// TIA Portal V20 export
// export: Created 2025-12-01T14:57:04.2343757Z, ExportSetting None, DisplayName Totally Integrated Automation Portal, DisplayVersion V20 Update 3, DisplayName TIA Portal Openness, DisplayVersion V20 Update 3, DisplayName TIA Portal Version Control Interface, DisplayVersion V20 Update 3, DisplayName STEP 7 Professional, DisplayVersion V20 Update 3, DisplayName STEP 7 Safety, DisplayVersion V20 Update 2, DisplayName WinCC Basic/Comfort/Advanced, DisplayVersion V20 Update 3, DisplayName WinCC Professional, DisplayVersion V20 Update 3, DisplayName WinCC Unified, DisplayVersion V20 Update 3
FUNCTION "FC772_Control_ElevadorDobleHorq" : Void   // FC772, STL
TITLE = Tracking de la Maquina Base
{ S7_Optimized_Access := 'FALSE' }
AUTHOR : TRACKING
NAME : 20141014
VERSION : 4.0
// - Inicializar
// - Recoger datos necesarios del Sistema
// 
// - Dispositivo Maquina
//   + Gestion de Estado
//   + Gestion de Control de Reset
//   + Gestion de Control de Paro Blando
//   + Gestion de Control de Errores
// 
// - Operaciones propias de la Maquina
// 
// - Cierre de protocolo de la Maquina
// - Actualizar datos del Sistema
// stored: AutoNumber false
   VAR_INPUT
      EstadoZonaMaquina : "EstadoZona";   // Estado de la Maquina (ZONA)
      EstadoZonaMesaH01 : "EstadoZona";   // Estado de la Mesa H1 (ZONA)
      EstadoZonaMesaH02 : "EstadoZona";   // Estado de la Mesa H2 (ZONA)
      MaxPisos : UInt;   // Numero Maximo Pisos
      H01_Habilitada : Bool;   // Permiso trabajo con Horquilla 1
      H02_Habilitada : Bool;   // Permiso trabajo con Horquilla 2
      MesaH01_Vacia : Bool;   // Estado Mesa Horquilla 1 Vacia
      MesaH01_Cargada : Bool;   // Estado Mesa Horquilla 1 Cargada
      MesaH02_Vacia : Bool;   // Estado Mesa Horquilla 2 Vacia
      MesaH02_Cargada : Bool;   // Estado Mesa Horquilla 1 Cargada
      OrdenMesaH01 : Bool;   // Orden Tracking Mesa Horquilla 01
      OrdenMesaH02 : Bool;   // Orden Tracking Mesa Horquilla 02
      MesaDestinoH01 : UInt;   // Mesa Destino para UT en Mesa Horquilla 1
      MesaDestinoH02 : UInt;   // Mesa Destino para UT en Mesa Horquilla 2
      NDB_AuxliarElevador : UInt;   // Numero de DB auxiliar elevador
      OrdenH01_Acabada : Bool;   // Orden ejecutada por la Horquilla 1
      OrdenH02_Acabada : Bool;   // Orden ejecutada por la Horquilla 2
      OrdenPasarAReposo : Bool;   // Orden Para posicionar el carro en posición reposo
      PisoDeReposo : UInt;   // Piso para posición reposo
   END_VAR
   VAR_IN_OUT
      Orden_Piso : UInt;   // Piso del Movimiento a Ejecutar
      OrdenH01_TipoMovi : UInt;   // Tipo de Movimiento a Ejecutar con la Horquilla 1
      OrdenH02_TipoMovi : UInt;   // Tipo de Movimeinto a Ejecutar con la Horquilla 2
      MesaEntrada_H01 : UInt;   // Mesa con Transferencia hacia la Horquilla 1
      MesaEntrada_H02 : UInt;   // Mesa con Transferencia hacia la Horquilla 2
      MesaSalida_H01 : UInt;   // Mesa con Transferencia desde la Horquilla 1
      MesaSalida_H02 : UInt;   // Mesa con Transferencia desde la Horquilla 2
      OrdenH01_Realizar : Bool;   // Orden de Ejecutar Movimiento para la Horquilla 2
      OrdenH02_Realizar : Bool;   // Orden de Ejecutar Movimiento para la Horquilla 1
      MemoriaPisoCarga : UInt;   // Memoriza Ultimo Piso Carga
      PisoUltimaOrden : UInt;   // Memoriza Piso de la Ultima Orden Enviada
   END_VAR
   VAR_TEMP
      DBAuxElevador : Word;
      DBTMPTracking : Word;   // Num. DB de los Temporizadores
      Maquina : UInt;   // Numero de Maquina dentro del PLC
      NumPisoDescarga : UInt;
      TempInt : UInt;
      SinUT : Bool;
   END_VAR
BEGIN

NETWORK
TITLE = Inicializar
// - Inicializar las Varriables
// - Inicializar para la Base de datos
// - Inicializar para las comunicaciones
/////////////////////////////////////////////////////////////////////////////
// --- Inicializar las Variables



NETWORK
TITLE = Reset de Variables
/////////////////////////////////////////////////////////////////////////////
// --- Si realiza un reset hay que limpiar las variables

      AN    #EstadoZonaMaquina.PerReset_CBx;
      JC    NoExiste_Reset;  // Reseteada la Maquina

      L     0;  // Reseteo de las Ordenes de las Horquillas
      T     #OrdenH01_TipoMovi;
      T     #OrdenH02_TipoMovi;
      R     #OrdenH01_Realizar;
      R     #OrdenH02_Realizar;

      L     0;  // Reseteo del Numero de Piso
      T     #Orden_Piso;

      L     0;  // Datos del Tracking
      T     #MesaEntrada_H01;  // del elevador de doble Horquilla
      T     #MesaEntrada_H02;
      T     #MesaSalida_H01;
      T     #MesaSalida_H02;

      JU    FinalFuncion;  // Finalizado el tratamiento de la Maquina

NoExiste_Reset:NOP   0;



NETWORK
TITLE = Elevador Doble (Particular del Tipo de Maquina)
/////////////////////////////////////////////////////////////////////////////
// ---
// ---           GENERAR ORDNES PARA EL ELEVADOR DOBLE
// ---
/////////////////////////////////////////////////////////////////////////////

      L     #NDB_AuxliarElevador;  // DB Auxliar del Elevador
      T     #DBAuxElevador;


/////////////////////////////////////////////////////////////////////////////
// --- No Ordernes y alguna Vacia, incrementar piso, para buscar AVISO

      AN    #OrdenH01_Realizar;  // No tiene Orden H01
      AN    #OrdenH02_Realizar;  // No tiene Orden H02
      A(;
      O     #MesaH01_Vacia;  // Una de las Horquillas este Vacia
      O     #MesaH02_Vacia;
      );
      JCN   ControlHorquillas;  // Si no cumple saltar a ver por horquilla


/////////////////////////////////////////////////////////////////////////////
// ---- Incremento de Busqueda de Pisos - Control de Pisos

      L     1;  // Se incrementa el Piso
      L     #MemoriaPisoCarga;
      +I;
      T     #MemoriaPisoCarga;

      L     #MemoriaPisoCarga;  // Si Piso > MaxPisos
      L     #MaxPisos;  // Inicializar Piso de Busqueda = 1
      >I;
      JC    IncializaPisoCarga;  // Si tiene que saltar a Inicializar Piso

      L     #MemoriaPisoCarga;  // Si Piso < 1
      L     1;  // Inicializar Piso de Busqueda = 1
      <I;
      JC    IncializaPisoCarga;  // Si tiene que saltar a Inicializar Piso

      JU    ControlHorquillas;  // Saltar a ver Horquillas

IncializaPisoCarga:L     0;  // Inicializar Piso
      T     #MemoriaPisoCarga;


/////////////////////////////////////////////////////////////////////////////
// --- Control a las Hoquillas
ControlHorquillas:NOP   0;



NETWORK
TITLE = Elevador Doble (Particular del Tipo de Maquina) - Horquilla 01
/////////////////////////////////////////////////////////////////////////////
// ---                CONTROL DE ORDENES PARA LA HORQUILLA 1
// ---
// ---  Si Horquilla No habilitada -> No se busca posible carga ni se mandan
// ---                             -> Ni se mandan Ordenes de Descarga
// ---  Si hay Orden en EJECUCION  -> Esperamos FIN EJECUCION
// ---
// ---  Si Mesa Cargada            -> Generar Orden de Descarga
// ---  Si Mesa Vacia              -> Generar Orden de Carga
// ---
/////////////////////////////////////////////////////////////////////////////

      SET;
      AN    #H01_Habilitada;  // Si Horquilla Habilitada
      JC    H1_Final;  // No hay que hacer nada con esta Horquilla

      SET;
      O     #OrdenH01_Realizar;  // Si hay Orden en EJECUCION
      O     #OrdenH01_Acabada;  // No acabado el cierre del Protocolo
      JC    H1_Final;  // Mirar si hay FIN EJECUCION

      SET;
      A     #MesaH01_Cargada;  // Si esta Cargada la Horquilla
      JC    DesCarga_H1;  // Ir a Mandar la Orden de Descarga

      SET;
      A     #MesaH01_Vacia;  // Esta Vacía la Hoquilla
      A     #OrdenMesaH01;  // Si Orden de Descarga H01
      JC    DesCarga_H1;  // Ir a Mandar la Orden de Descarga

      SET;
      A     #MesaH01_Vacia;  // Esta Vacía la Hoquilla
      JC    Carga_H1;  // Ir a Mandar la Orden de Carga

      JU    H1_Final;  // Por ahora no hacer nada



/////////////////////////////////////////////////////////////////////////////
/////////////////////////////////////////////////////////////////////////////
/////////////////////////////////////////////////////////////////////////////
/////////////////////////////////////////////////////////////////////////////
// ---                         ORDEN DE CARGA
// --- La Horquilla H01 esta Vacia -> Mirar si hay AVISO
// --- Se mira quee Piso dependiendo de hay Orden en H02

Carga_H1:NOP   0;
      AN    #OrdenH02_Realizar;  // Si hay Orden en H02, en CURSO ?
      JC    BusquedaPiso_DeOrdenCarga_H1;

      L     #Orden_Piso;  // Coger el Piso
      T     #MemoriaPisoCarga;  // De la Orden de la H02


/////////////////////////////////////////////////////////////////////////////
// --- BUSQUEDA de ver si hay ORDEN de CARGA en el Piso
BusquedaPiso_DeOrdenCarga_H1:NOP   0;

// --- Inicializar DB, Puntero y Variables

      L     #MemoriaPisoCarga;  // Puntero al Datos del Piso
      L     16;  // Longitud 16 Bytes
      *I;
      SLD   3;
      LAR2;

      L     0;  // Inicializar
      T     #OrdenH01_TipoMovi;  // Tipo de Movimiento
      T     #MesaEntrada_H01;  // Mesa de Entrada de la H1



/////////////////////////////////////////////////////////////////////////////
// --- Mirar si hay Orden de CARGA H01 para la Horquilla 1
// --- Condiciones para la H01 - Posibilidad de Carga Si:
// ---    + Preferencia de Carga, si Mesa H02 Vacia
// ---    + Mesa H02 cargada
// ---    + Realiazndo Orden en la H2
// ---    + Mesa H02 Desabilitada
// --- ANULAR POR AHORA 25/09/2012

//      U(
//      U     #MesaH02_Vacia              // Con la H02 Vacia, ver Si
//      AUF   DB [#DBAuxElevador]
//      U     DBX [AR2,P#14.2]            // Preferente H01 - Posicion 14.2

//      O     #MesaH02_Cargada            // Si la H02 esta Cargada
//      O     #OrdenH02_Realizar          // Si la H02 esta Realizando Orden
//      ON    #H02_Habilitada             // Si H02 No Habilitada
//      )
//      SPBN  H1_F                        // No se puede hacer ?

// --- Mirar si hay AVISO de la Carga

      OPN   DB [#DBAuxElevador];
      A     DBX [AR2, P#14.0];  // Acceso OK    - Pos 14.0
      A     DBX [AR2, P#0.0];  // AVISO Carga  - Pos 0.0
      JC    OrdenCarga_H1Derecha;  // Orden de Carga a la Derecha

      OPN   DB [#DBAuxElevador];
      A     DBX [AR2, P#14.0];  // Acceso OK    - Pos 14.0
      A     DBX [AR2, P#0.4];  // AVISO Carga  - Pos 0.4
      JC    OrdenCarga_H1Izquierda;  // Orden de Carga a la Izquierda

      JU    H1_Final;  // No más posibilidades de carga

/////////////////////////////////////////////////////////////////////////////
// --- Mandar la Orden de CARGA de la H01 por la Derecha

OrdenCarga_H1Derecha:NOP   0;
      L     W#16#25;  // TipoMov: Carga Simple Derecha
      T     #OrdenH01_TipoMovi;
      L     #MemoriaPisoCarga;  // Piso
      T     #Orden_Piso;
      T     #PisoUltimaOrden;

      SET;
      S     #OrdenH01_Realizar;  // Activaccion

      OPN   DB [#DBAuxElevador];
      L     DBW [AR2, P#6.0];  // Tracking - Posicion 6
      T     #MesaEntrada_H01;  // Mesa de Entrada de la H1

      JU    H1_Final;


/////////////////////////////////////////////////////////////////////////////
// --- Mandar la Orden de CARGA de la H01 por la Derecha

OrdenCarga_H1Izquierda:NOP   0;
      L     W#16#15;  // TipoMov: Carga,Simple,Izquierda
      T     #OrdenH01_TipoMovi;
      L     #MemoriaPisoCarga;  // Piso
      T     #Orden_Piso;
      T     #PisoUltimaOrden;

      SET;
      S     #OrdenH01_Realizar;  // Activaccion

      OPN   DB [#DBAuxElevador];
      L     DBW [AR2, P#8.0];  // Tracking - Posicion 8
      T     #MesaEntrada_H01;  // Mesa de Entrada de la H1

      JU    H1_Final;


// ---              FIN de las Casos de ORDEN de CARGA
/////////////////////////////////////////////////////////////////////////////
/////////////////////////////////////////////////////////////////////////////



/////////////////////////////////////////////////////////////////////////////
// --- Mirar si hay Orden de DESCARGA H01 para la Horquilla 1
// ---    + Mirar si hay Orden de Descarga para la H1
// ---    + Buscar Piso

DesCarga_H1:AN    #OrdenMesaH01;  // Si Orden de Descarga H01
      JC    H1_Final;


// --- Mesa Destino debe estar Vacia antes de Enviar la Orden

      L     #MesaDestinoH01;  // Paso la Variable a Entero
      T     #TempInt;

      CALL  "FC870_MesaSinUT"
      ( Mesa  := #TempInt,
        SinUT := #SinUT
      );  // Mirar si Mesa Destino esta Vacia

      AN    #SinUT;
      JC    H1_Final;  // Esta vacia ?

// --- Inicializar Variables

      L     0;  // Inicializar
      T     #OrdenH01_TipoMovi;  // Tipo de Movimiento
      T     #MesaSalida_H01;  // Mesa de Destino de la H1

// --- Buscar el Piso de Descarga

      L     1;  // Empiezo la Busqueda
      T     #NumPisoDescarga;  // Por el Piso 01

BusquedaPiso_DeOrdenDescarga_H1:NOP   0;
      L     #NumPisoDescarga;  // Puntero de Piso
      L     16;  // Longitud 16 Bytes
      *I;
      SLD   3;
      LAR2;

      OPN   DB [#DBAuxElevador];
      L     DBW [AR2, P#6.0];  // Mesa_Derecha - Posicion 6
      L     #MesaDestinoH01;  // Mesa Destino de la Orden
      ==I;
      JC    OrdenDesCarga_H1Derecha;  // Es Mesa de Salida Derecha ?

      OPN   DB [#DBAuxElevador];
      L     DBW [AR2, P#8.0];  // Mesa Izquierda - Posicion 8
      L     #MesaDestinoH01;  // Mesa Destino de la Orden
      ==I;
      JC    OrdenDesCarga_H1Izquierda;  // Mesa Izquierda de Salida

      L     1;  // Aumentar de Piso
      L     #NumPisoDescarga;  // Para ver el Siguiente
      +I;
      T     #NumPisoDescarga;

      L     #NumPisoDescarga;
      L     #MaxPisos;
      <=I;
      JC    BusquedaPiso_DeOrdenDescarga_H1;  // Todavia quedan pisos por Buscar

// --- No se encuentra piso para enviar el piso de Descarga
// --- Hay algun error en la ruta ¿QUE HACER?

      JU    H1_Final;


/////////////////////////////////////////////////////////////////////////////
// --- Mandar Orden de DESCARGA de la Hoquilla 1 por la Derecha

OrdenDesCarga_H1Derecha:NOP   0;
      A     #OrdenH02_Realizar;  // Si H02 Realizando Orden
      A(;  // Debe ser el mismo Piso Destino
      L     #NumPisoDescarga;
      L     #Orden_Piso;
      <>I;
      );
      JC    H1_Final;

      L     W#16#29;  // TipoMov: Descarga,Simple,Derecha
      T     #OrdenH01_TipoMovi;
      L     #NumPisoDescarga;  // Piso
      T     #Orden_Piso;
      T     #PisoUltimaOrden;

      SET;
      S     #OrdenH01_Realizar;  // Activacion de la Orden

      L     #MesaDestinoH01;
      T     #MesaSalida_H01;  // Mesa de Destino de la H1

      JU    H1_Final;


/////////////////////////////////////////////////////////////////////////////
// --- Mandar Orden de DESCARGA de la Hoquilla 1 por la Izquierda

OrdenDesCarga_H1Izquierda:NOP   0;
      A     #OrdenH02_Realizar;  // Si H02 Realizando Orden
      A(;  // Debe ser el mismo Piso Destino
      L     #NumPisoDescarga;
      L     #Orden_Piso;
      <>I;
      );
      JC    H1_Final;

      L     W#16#19;  // TipoMov: Descarga,Simple,Izquierda
      T     #OrdenH01_TipoMovi;
      L     #NumPisoDescarga;  // Piso
      T     #Orden_Piso;
      T     #PisoUltimaOrden;

      SET;
      S     #OrdenH01_Realizar;  // Activacion de la Orden

      L     #MesaDestinoH01;
      T     #MesaSalida_H01;  // Mesa de Destino de la H1

      JU    H1_Final;


// ---              FIN de las Casos de ORDEN de DESCARGA
/////////////////////////////////////////////////////////////////////////////
/////////////////////////////////////////////////////////////////////////////




/////////////////////////////////////////////////////////////////////////////
// --- Final del CONTROL de Ordenes para la HORQUILLA 1
// --- Cierre del PROTOCOLO de EJECUCION

H1_Final:NOP   0;
      A     #OrdenH01_Realizar;
      A     #OrdenH01_Acabada;
      JCN   FinTratamiento_H1;

      L     0;  // Reseteo para la Orden de la H01
      T     #OrdenH01_TipoMovi;
      T     #MesaEntrada_H01;
      T     #MesaSalida_H01;

      SET;
      R     #OrdenH01_Realizar;


/////////////////////////////////////////////////////////////////////////////
// --- Final para la Horquilla 1
FinTratamiento_H1:NOP   0;



NETWORK
TITLE = Elevador Doble (Particular del Tipo de Maquina) - Horquilla 02
/////////////////////////////////////////////////////////////////////////////
// ---                CONTROL DE ORDENES PARA LA HORQUILLA 2
// ---
// ---  Si Horquilla No habilitada -> No se busca posible carga ni se mandan
// ---                             -> Ni se mandan Ordenes de Descarga
// ---  Si hay Orden en EJECUCION  -> Esperamos FIN EJECUCION
// ---
// ---  Si Mesa Cargada            -> Generar Orden de Descarga
// ---  Si Mesa Vacia              -> Generar Orden de Carga
// ---
/////////////////////////////////////////////////////////////////////////////

      SET;
      AN    #H02_Habilitada;  // Si Horquilla Habilitada
      JC    H2_Final;  // No hay que hacer nada con esta Horquilla

      SET;
      O     #OrdenH02_Realizar;  // Si hay Orden en EJECUCION
      O     #OrdenH01_Acabada;  // No acabado el cierre del Protocolo
      JC    H2_Final;  // Mirar si hay FIN EJECUCION

      SET;
      A     #MesaH02_Cargada;  // Si esta Cargada la Horquilla
      JC    DesCarga_H2;  // Ir a Mandar la Orden de Descarga

      SET;
      A     #MesaH02_Vacia;  // Esta Vacía la Hoquilla
      A     #OrdenMesaH02;  // Si Orden de Descarga H02
      JC    DesCarga_H2;  // Ir a Mandar la Orden de Descarga

      SET;
      A     #MesaH02_Vacia;  // Esta Vacía la Hoquilla
      JC    Carga_H2;  // Ir a Mandar la Orden de Carga

      JU    H2_Final;  // Por ahora no hacer nada




/////////////////////////////////////////////////////////////////////////////
// ---                         ORDEN DE CARGA
// --- La Horquilla H02 esta Vacia -> Mirar si hay AVISO
// --- Se mira quee Piso dependiendo de hay Orden en H01

Carga_H2:NOP   0;
      SET;
      AN    #OrdenH01_Realizar;  // Si hay Orden en H01, en CURSO ?
      JC    BusquedaPiso_DeOrdenCarga_H2;

      L     #Orden_Piso;  // Coger el Piso
      T     #MemoriaPisoCarga;  // De la Orden de la H01

/////////////////////////////////////////////////////////////////////////////
// --- BUSQUEDA de ver si hay ORDEN de CARGA en el Piso
// ---  * Inicializar DB, Puntero y Variables

BusquedaPiso_DeOrdenCarga_H2:NOP   0;
      L     #MemoriaPisoCarga;  // Puntero al Datos del Piso
      L     16;  // Longitud 16 Bytes
      *I;
      SLD   3;
      LAR2;

      L     0;  // Inicializar
      T     #OrdenH02_TipoMovi;  // Tipo de Movimiento
      T     #MesaEntrada_H02;  // Mesa de Entrada de H2

/////////////////////////////////////////////////////////////////////////////
// --- Mirar si hay Orden de CARGA H02 para la Horquilla 2
// --- Condiciones para la H02 - Posibilidad de Carga Si:
// ---    + Preferencia de Carga, si Mesa H01 Vacia
// ---    + Mesa H01 cargada
// ---    + Realizndo Orden en la H1
// ---    + Mesa H01 Desabilitada
// --- ANULAR POR AHORA 25/09/2012

//      U(
//      U     #MesaH01_Vacia              // Con la H01 Vacia, ver Si
//      AUF   DB [#DBAuxElevador]
//      U     DBX [AR2,P#14.3]            // Preferente H02 - Posicion 14.3

//      O     #MesaH01_Cargada            // Si la H01 esta Cargada
//      O     #OrdenH01_Realizar          // Si la H01 esta Realizando Orden
//      ON    #H01_Habilitada             // Si H01 No Habilitada
//      )
//      SPBN  H2_F                        // No se puede hacer ?

// --- Mirar si hay AVISO de Carga

      OPN   DB [#DBAuxElevador];
      A     DBX [AR2, P#14.1];  // Acceso OK    - Pos 14.1
      A     DBX [AR2, P#2.0];  // AVISO Carga  - Pos 2.0
      JC    OrdenCarga_H2Derecha;  // Orden de Carga a la Derecha

      OPN   DB [#DBAuxElevador];
      A     DBX [AR2, P#14.1];  // Acceso OK    - Pos 14.1
      A     DBX [AR2, P#2.4];  // AVISO Carga  - Pos 2.4
      JC    OrdenCarga_H2Izquierda;  // Orden de Carga a la Izquierda

      JU    H2_Final;  // No más posibilidades de carga


/////////////////////////////////////////////////////////////////////////////
// --- Mandar la Orden de CARGA de la H01 por la Derecha

OrdenCarga_H2Derecha:NOP   0;
      L     W#16#25;  // TipoMov: Carga Simple Derecha
      T     #OrdenH02_TipoMovi;
      L     #MemoriaPisoCarga;  // Piso
      T     #Orden_Piso;
      T     #PisoUltimaOrden;

      SET;
      S     #OrdenH02_Realizar;  // Activaccion

      OPN   DB [#DBAuxElevador];
      L     DBW [AR2, P#10.0];  // Tracking - Posicion 10
      T     #MesaEntrada_H02;  // Mesa de Entrada de la H2

      JU    H2_Final;


/////////////////////////////////////////////////////////////////////////////
// --- Mandar la Orden de CARGA de la H01 por la Derecha

OrdenCarga_H2Izquierda:NOP   0;
      L     W#16#15;  // TipoMov: Carga,Simple,Izquierda
      T     #OrdenH02_TipoMovi;
      L     #MemoriaPisoCarga;  // Piso
      T     #Orden_Piso;
      T     #PisoUltimaOrden;

      SET;
      S     #OrdenH02_Realizar;  // Activaccion

      OPN   DB [#DBAuxElevador];
      L     DBW [AR2, P#12.0];  // Tracking - Posicion 12
      T     #MesaEntrada_H02;  // Mesa de Entrada de la H2

      JU    H2_Final;


// ---              FIN de las Casos de ORDEN de CARGA
/////////////////////////////////////////////////////////////////////////////
/////////////////////////////////////////////////////////////////////////////
/////////////////////////////////////////////////////////////////////////////




/////////////////////////////////////////////////////////////////////////////
/////////////////////////////////////////////////////////////////////////////
/////////////////////////////////////////////////////////////////////////////
// --- Mirar si hay Orden de DESCARGA H02 para la Horquilla 2
// ---    + Mirar si hay Orden de Descarga para la H2
// ---    + Buscar Piso

DesCarga_H2:NOP   0;
      SET;
      AN    #OrdenMesaH02;  // Si Orden de Descarga H02
      JC    H2_Final;

// --- Mesa Destino debe estar Vacia antes de Enviar la Orden

      L     #MesaDestinoH02;  // Paso la Variable a Entero
      T     #TempInt;

      CALL  "FC870_MesaSinUT"
      ( Mesa  := #TempInt,
        SinUT := #SinUT
      );  // Mirar si Mesa Destino esta Vacia

      AN    #SinUT;
      JC    H2_Final;  // Esta vacia ?

// --- Inicializar

      L     0;  // Inicializar
      T     #OrdenH02_TipoMovi;  // Tipo de Movimiento
      T     #MesaSalida_H02;  // Mesa de Destino de la H2

// --- Buscar el Piso de Descarga

      L     1;  // Empiezo la Busqueda
      T     #NumPisoDescarga;  // Por el Piso 01

BusquedaPiso_DeOrdenDescarga_H2:NOP   0;
      L     #NumPisoDescarga;  // Puntero de Piso
      L     16;  // Longitud 16 Bytes
      *I;
      SLD   3;
      LAR2;

      OPN   DB [#DBAuxElevador];
      L     DBW [AR2, P#10.0];  // Mesa_Derecha - Posicion 10
      L     #MesaDestinoH02;  // Mesa Destino de la Orden
      ==I;
      JC    OrdenDesCarga_H2Derecha;  // Es Mesa de Salida Derecha ?

      OPN   DB [#DBAuxElevador];
      L     DBW [AR2, P#12.0];  // Mesa Izquierda - Posicion 12
      L     #MesaDestinoH02;  // Mesa Destino de la Orden
      ==I;
      JC    OrdenDesCarga_H2Izquierda;  // Mesa Izquierda de Salida

      L     1;  // Aumentar de Piso
      L     #NumPisoDescarga;  // Para ver el Siguiente
      +I;
      T     #NumPisoDescarga;

      L     #NumPisoDescarga;
      L     #MaxPisos;
      <=I;
      JC    BusquedaPiso_DeOrdenDescarga_H2;  // Todavia quedan pisos por Buscar

// --- No se encuentra piso para enviar el piso de Descarga
// --- Hay algun error en la ruta ¿QUE HACER?

      JU    H2_Final;

/////////////////////////////////////////////////////////////////////////////
// --- Mandar Orden de DESCARGA de la Hoquilla 2 por la Derecha

OrdenDesCarga_H2Derecha:NOP   0;
      A     #OrdenH01_Realizar;  // Si H01 Realizando Orden
      A(;  // Debe ser el mismo Piso Destino
      L     #NumPisoDescarga;
      L     #Orden_Piso;
      <>I;
      );
      JC    H2_Final;

      L     W#16#29;  // TipoMov: Descarga,Simple,Derecha
      T     #OrdenH02_TipoMovi;
      L     #NumPisoDescarga;  // Piso
      T     #Orden_Piso;
      T     #PisoUltimaOrden;

      SET;
      S     #OrdenH02_Realizar;  // Activacion de la Orden

      L     #MesaDestinoH02;
      T     #MesaSalida_H02;  // Mesa de Destino de la H2

      JU    H2_Final;

/////////////////////////////////////////////////////////////////////////////
// --- Mandar Orden de DESCARGA de la Hoquilla 2 por la Izquierda

OrdenDesCarga_H2Izquierda:NOP   0;
      A     #OrdenH01_Realizar;  // Si H01 Realizando Orden
      A(;  // Debe ser el mismo Piso Destino
      L     #NumPisoDescarga;
      L     #Orden_Piso;
      <>I;
      );
      JC    H2_Final;

      L     W#16#19;  // TipoMov: Descarga,Simple,Izquierda
      T     #OrdenH02_TipoMovi;
      L     #NumPisoDescarga;  // Piso
      T     #Orden_Piso;
      T     #PisoUltimaOrden;

      SET;
      S     #OrdenH02_Realizar;  // Activacion de la Orden

      L     #MesaDestinoH02;
      T     #MesaSalida_H02;  // Mesa de Destino de la H2

      JU    H2_Final;


// ---              FIN de las Casos de ORDEN de DESCARGA
/////////////////////////////////////////////////////////////////////////////
/////////////////////////////////////////////////////////////////////////////
/////////////////////////////////////////////////////////////////////////////




/////////////////////////////////////////////////////////////////////////////
// --- Final del CONTROL de Ordenes para la HORQUILLA 2
// --- Cierre del PROTOCOLO de EJECUCION

H2_Final:NOP   0;
      SET;
      A     #OrdenH02_Realizar;
      A     #OrdenH02_Acabada;
      JCN   FinTratamiento_H2;

      L     0;  // Reseteo para la Orden de la H02
      T     #OrdenH02_TipoMovi;
      T     #MesaEntrada_H02;
      T     #MesaSalida_H02;

      SET;
      R     #OrdenH02_Realizar;


/////////////////////////////////////////////////////////////////////////////
// --- Final para la Horquilla 1
FinTratamiento_H2:NOP   0;



NETWORK
TITLE = Elevador Doble (Particular del Tipo de Maquina) - Comun de Horq
/////////////////////////////////////////////////////////////////////////////
// --- Reseteo de los numero de Piso, comun a las dos Horquillas

      SET;
      AN    #OrdenH01_Realizar;
      AN    #OrdenH02_Realizar;
      JCN   FinComunicaHorquilla;

      L     0;
      T     #Orden_Piso;

FinComunicaHorquilla:NOP   0;



NETWORK
TITLE = Elevador Doble (Particular del Tipo de Maquina) - Paso a Reposo
/////////////////////////////////////////////////////////////////////////////
// ---                      PASAR A REPOSO
// ---  Se Mandara siempre para la  Horquilla 1
// ---  Si Mesas Vacias, sin Orden  y Orden Posicionar Activar Orden en H1
// ---  Tiene que cumplir siempre estas Condiciones:
// ---      + Horquillas Vacias
// ---      + Horquillas Sin Orden
// ---      + Y tener orden de ir a Reposo

      SET;
//     U     #MesaH01_Vacia       // Estan Vacias
//     U     #MesaH02_Vacia
      AN    #OrdenH01_Realizar;  // Estan sin Orden
      AN    #OrdenH02_Realizar;
      AN    #OrdenH01_Acabada;
      AN    #OrdenH02_Acabada;
      A     #OrdenPasarAReposo;  // Orden de Pasar a Reposo
      JCN   Final_PasarReposo;  // Si no se cumple

      L     W#16#C;  // TipoMov: Posicionar
      T     #OrdenH01_TipoMovi;
      L     #PisoDeReposo;  // Piso de Reposo
      T     #Orden_Piso;

      SET;
      S     #OrdenH01_Realizar;  // Activacion


/////////////////////////////////////////////////////////////////////////////
// --- Final de PASAR A REPOSO
Final_PasarReposo:NOP   0;



NETWORK
TITLE = Final de la Funcion
/////////////////////////////////////////////////////////////////////////////
// --- Final de la funcion
FinalFuncion:NOP   0;


END_FUNCTION
